   cmAnodeNgBoxLiftUpDown.monitoring.error := FALSE;
   cmAnodeNgBoxLiftUpDown.monitoring.interlockHomePos := TRUE;
   cmAnodeNgBoxLiftUpDown.monitoring.interlockWorkPos := TRUE;
   cmAnodeNgBoxLiftUpDown.monitoring.status := 16#7006;
   cmAnodeNgBoxLiftUpDown.monitoring.interlockWarningWorkPos := FALSE;
   cmAnodeNgBoxLiftUpDown.monitoring.interlockWarningHomePos := FALSE;
   cmAnodeNgBoxLiftUpDown.configuration.referenceDesignator := WSTRING#'TwoWayAct.';
   cmAnodeNgBoxLiftUpDown.configuration.monitoringLeavingFeedback := T#5S;
   cmAnodeNgBoxLiftUpDown.configuration.monitoringReachingFeedback := T#5S;
   cmAnodeNgBoxLiftUpDown.configuration.monitoringDiscrepancy := T#0MS;
   cmAnodeNgBoxLiftUpDown.configuration.setOutputHomeContinuously := TRUE;
   cmAnodeNgBoxLiftUpDown.configuration.setOutputWorkContinuously := TRUE;
   cmAnodeNgBoxLiftUpDown.configuration.disableHomeCommand := FALSE;
   cmAnodeNgBoxLiftUpDown.configuration.disableFeedbackHomePos := FALSE;
   cmAnodeNgBoxLiftUpDown.configuration.disableFeedbackWorkPos := FALSE;
   cmAnodeNgBoxLiftUpDown.configuration.disableAlarms := FALSE;
   cmAnodeNgBoxLiftUpDown.configuration.resetOutputsOnError := FALSE;
   cmAnodeNgBoxLiftUpDown.configuration.allwaysWaitOnReachingTime := FALSE;
   cmAnodeNgBoxLockUpDown.commands.refreshConfiguration := FALSE;
   cmAnodeNgBoxLockUpDown.commands.editConfiguration := FALSE;
   cmAnodeNgBoxLockUpDown.commands.saveConfiguration := FALSE;
   cmAnodeNgBoxLockUpDown.commands.reset := FALSE;
   cmAnodeNgBoxLockUpDown.commands.commandHomePos := FALSE;
   cmAnodeNgBoxLockUpDown.commands.commandWorkPos := FALSE;
   cmAnodeNgBoxLockUpDown.monitoring.enable := TRUE;
   cmAnodeNgBoxLockUpDown.monitoring.referenceDesignator := WSTRING#'NgBoxLockUpDown';
   cmAnodeNgBoxLockUpDown.monitoring.commandHomePos := FALSE;
   cmAnodeNgBoxLockUpDown.monitoring.commandWorkPos := FALSE;
   cmAnodeNgBoxLockUpDown.monitoring.goToHomePos := FALSE;
   cmAnodeNgBoxLockUpDown.monitoring.goToWorkPos := FALSE;
   cmAnodeNgBoxLockUpDown.monitoring.inHomePos := FALSE;
   cmAnodeNgBoxLockUpDown.monitoring.inWorkPos := FALSE;
   cmAnodeNgBoxLockUpDown.monitoring.reset := FALSE;
   cmAnodeNgBoxLockUpDown.monitoring.enableManualCmds := FALSE;
   cmAnodeNgBoxLockUpDown.monitoring.error := FALSE;
   cmAnodeNgBoxLockUpDown.monitoring.interlockHomePos := TRUE;
   cmAnodeNgBoxLockUpDown.monitoring.interlockWorkPos := TRUE;
   cmAnodeNgBoxLockUpDown.monitoring.status := 16#7003;
   cmAnodeNgBoxLockUpDown.monitoring.interlockWarningWorkPos := FALSE;
   cmAnodeNgBoxLockUpDown.monitoring.interlockWarningHomePos := FALSE;
   cmAnodeNgBoxLockUpDown.configuration.referenceDesignator := WSTRING#'TwoWayAct.';
   cmAnodeNgBoxLockUpDown.configuration.monitoringLeavingFeedback := T#5S;
   cmAnodeNgBoxLockUpDown.configuration.monitoringReachingFeedback := T#5S;
   cmAnodeNgBoxLockUpDown.configuration.monitoringDiscrepancy := T#0MS;
   cmAnodeNgBoxLockUpDown.configuration.setOutputHomeContinuously := TRUE;
   cmAnodeNgBoxLockUpDown.configuration.setOutputWorkContinuously := TRUE;
   cmAnodeNgBoxLockUpDown.configuration.disableHomeCommand := FALSE;
   cmAnodeNgBoxLockUpDown.configuration.disableFeedbackHomePos := FALSE;
   cmAnodeNgBoxLockUpDown.configuration.disableFeedbackWorkPos := FALSE;
   cmAnodeNgBoxLockUpDown.configuration.disableAlarms := FALSE;
   cmAnodeNgBoxLockUpDown.configuration.resetOutputsOnError := FALSE;
   cmAnodeNgBoxLockUpDown.configuration.allwaysWaitOnReachingTime := FALSE;
   cmAnodeNgPnpVaccum.commands.refreshConfiguration := FALSE;
   cmAnodeNgPnpVaccum.commands.editConfiguration := FALSE;
   cmAnodeNgPnpVaccum.commands.saveConfiguration := FALSE;
   cmAnodeNgPnpVaccum.commands.reset := FALSE;
   cmAnodeNgPnpVaccum.commands.commandHomePos := FALSE;
   cmAnodeNgPnpVaccum.commands.commandWorkPos := FALSE;
   cmAnodeNgPnpVaccum.monitoring.enable := TRUE;
   cmAnodeNgPnpVaccum.monitoring.referenceDesignator := WSTRING#'NgPnpVaccum';
   cmAnodeNgPnpVaccum.monitoring.commandHomePos := FALSE;
   cmAnodeNgPnpVaccum.monitoring.commandWorkPos := FALSE;
   cmAnodeNgPnpVaccum.monitoring.goToHomePos := FALSE;
   cmAnodeNgPnpVaccum.monitoring.goToWorkPos := FALSE;
   cmAnodeNgPnpVaccum.monitoring.inHomePos := TRUE;
   cmAnodeNgPnpVaccum.monitoring.inWorkPos := FALSE;
   cmAnodeNgPnpVaccum.monitoring.reset := FALSE;
   cmAnodeNgPnpVaccum.monitoring.enableManualCmds := FALSE;
   cmAnodeNgPnpVaccum.monitoring.error := FALSE;
   cmAnodeNgPnpVaccum.monitoring.interlockHomePos := TRUE;
   cmAnodeNgPnpVaccum.monitoring.interlockWorkPos := TRUE;
   cmAnodeNgPnpVaccum.monitoring.status := 16#7003;
   cmAnodeNgPnpVaccum.monitoring.interlockWarningWorkPos := FALSE;
   cmAnodeNgPnpVaccum.monitoring.interlockWarningHomePos := FALSE;
   cmAnodeNgPnpVaccum.configuration.referenceDesignator := WSTRING#'TwoWayAct.';
   cmAnodeNgPnpVaccum.configuration.monitoringLeavingFeedback := T#5S;
   cmAnodeNgPnpVaccum.configuration.monitoringReachingFeedback := T#5S;
   cmAnodeNgPnpVaccum.configuration.monitoringDiscrepancy := T#0MS;
   cmAnodeNgPnpVaccum.configuration.setOutputHomeContinuously := TRUE;
   cmAnodeNgPnpVaccum.configuration.setOutputWorkContinuously := TRUE;
   cmAnodeNgPnpVaccum.configuration.disableHomeCommand := FALSE;
   cmAnodeNgPnpVaccum.configuration.disableFeedbackHomePos := FALSE;
   cmAnodeNgPnpVaccum.configuration.disableFeedbackWorkPos := FALSE;
   cmAnodeNgPnpVaccum.configuration.disableAlarms := FALSE;
   cmAnodeNgPnpVaccum.configuration.resetOutputsOnError := FALSE;
   cmAnodeNgPnpVaccum.configuration.allwaysWaitOnReachingTime := FALSE;
   cmAnodeConveyorCoverFwdBwd.commands.refreshConfiguration := FALSE;
   cmAnodeConveyorCoverFwdBwd.commands.editConfiguration := FALSE;
   cmAnodeConveyorCoverFwdBwd.commands.saveConfiguration := FALSE;
   cmAnodeConveyorCoverFwdBwd.commands.reset := FALSE;
   cmAnodeConveyorCoverFwdBwd.commands.commandHomePos := FALSE;
   cmAnodeConveyorCoverFwdBwd.commands.commandWorkPos := FALSE;
   cmAnodeConveyorCoverFwdBwd.monitoring.enable := TRUE;
   cmAnodeConveyorCoverFwdBwd.monitoring.referenceDesignator := WSTRING#'ConveyorCoverFwdBwd';
   cmAnodeConveyorCoverFwdBwd.monitoring.commandHomePos := FALSE;
   cmAnodeConveyorCoverFwdBwd.monitoring.commandWorkPos := FALSE;
   cmAnodeConveyorCoverFwdBwd.monitoring.goToHomePos := FALSE;
   cmAnodeConveyorCoverFwdBwd.monitoring.goToWorkPos := FALSE;
   cmAnodeConveyorCoverFwdBwd.monitoring.inHomePos := FALSE;
   cmAnodeConveyorCoverFwdBwd.monitoring.inWorkPos := FALSE;
   cmAnodeConveyorCoverFwdBwd.monitoring.reset := FALSE;
   cmAnodeConveyorCoverFwdBwd.monitoring.enableManualCmds := FALSE;
   cmAnodeConveyorCoverFwdBwd.monitoring.error := FALSE;
   cmAnodeConveyorCoverFwdBwd.monitoring.interlockHomePos := TRUE;
   cmAnodeConveyorCoverFwdBwd.monitoring.interlockWorkPos := TRUE;
   cmAnodeConveyorCoverFwdBwd.monitoring.status := 16#7003;
   cmAnodeConveyorCoverFwdBwd.monitoring.interlockWarningWorkPos := FALSE;
   cmAnodeConveyorCoverFwdBwd.monitoring.interlockWarningHomePos := FALSE;
   cmAnodeConveyorCoverFwdBwd.configuration.referenceDesignator := WSTRING#'TwoWayAct.';
   cmAnodeConveyorCoverFwdBwd.configuration.monitoringLeavingFeedback := T#5S;
   cmAnodeConveyorCoverFwdBwd.configuration.monitoringReachingFeedback := T#5S;
   cmAnodeConveyorCoverFwdBwd.configuration.monitoringDiscrepancy := T#0MS;
   cmAnodeConveyorCoverFwdBwd.configuration.setOutputHomeContinuously := TRUE;
   cmAnodeConveyorCoverFwdBwd.configuration.setOutputWorkContinuously := TRUE;
   cmAnodeConveyorCoverFwdBwd.configuration.disableHomeCommand := FALSE;
   cmAnodeConveyorCoverFwdBwd.configuration.disableFeedbackHomePos := FALSE;
   cmAnodeConveyorCoverFwdBwd.configuration.disableFeedbackWorkPos := FALSE;
   cmAnodeConveyorCoverFwdBwd.configuration.disableAlarms := FALSE;
   cmAnodeConveyorCoverFwdBwd.configuration.resetOutputsOnError := FALSE;
   cmAnodeConveyorCoverFwdBwd.configuration.allwaysWaitOnReachingTime := FALSE;
   cmAnodeConveyorPickUpBlower.commands.refreshConfiguration := FALSE;
   cmAnodeConveyorPickUpBlower.commands.editConfiguration := FALSE;
   cmAnodeConveyorPickUpBlower.commands.saveConfiguration := FALSE;
   cmAnodeConveyorPickUpBlower.commands.reset := FALSE;
   cmAnodeConveyorPickUpBlower.commands.commandHomePos := FALSE;
   cmAnodeConveyorPickUpBlower.commands.commandWorkPos := FALSE;
   cmAnodeConveyorPickUpBlower.monitoring.enable := TRUE;
   cmAnodeConveyorPickUpBlower.monitoring.referenceDesignator := WSTRING#'ConveyorPickUpBlower';
   cmAnodeConveyorPickUpBlower.monitoring.commandHomePos := FALSE;
   cmAnodeConveyorPickUpBlower.monitoring.commandWorkPos := FALSE;
   cmAnodeConveyorPickUpBlower.monitoring.goToHomePos := FALSE;
   cmAnodeConveyorPickUpBlower.monitoring.goToWorkPos := TRUE;
   cmAnodeConveyorPickUpBlower.monitoring.inHomePos := FALSE;
   cmAnodeConveyorPickUpBlower.monitoring.inWorkPos := TRUE;
   cmAnodeConveyorPickUpBlower.monitoring.reset := FALSE;
   cmAnodeConveyorPickUpBlower.monitoring.enableManualCmds := FALSE;
   cmAnodeConveyorPickUpBlower.monitoring.error := FALSE;
   cmAnodeConveyorPickUpBlower.monitoring.interlockHomePos := TRUE;
   cmAnodeConveyorPickUpBlower.monitoring.interlockWorkPos := TRUE;
   cmAnodeConveyorPickUpBlower.monitoring.status := 16#7006;
   cmAnodeConveyorPickUpBlower.monitoring.interlockWarningWorkPos := FALSE;
   cmAnodeConveyorPickUpBlower.monitoring.interlockWarningHomePos := FALSE;
   cmAnodeConveyorPickUpBlower.configuration.referenceDesignator := WSTRING#'TwoWayAct.';
   cmAnodeConveyorPickUpBlower.configuration.monitoringLeavingFeedback := T#5S;
   cmAnodeConveyorPickUpBlower.configuration.monitoringReachingFeedback := T#5S;
   cmAnodeConveyorPickUpBlower.configuration.monitoringDiscrepancy := T#0MS;
   cmAnodeConveyorPickUpBlower.configuration.setOutputHomeContinuously := TRUE;
   cmAnodeConveyorPickUpBlower.configuration.setOutputWorkContinuously := TRUE;
   cmAnodeConveyorPickUpBlower.configuration.disableHomeCommand := FALSE;
   cmAnodeConveyorPickUpBlower.configuration.disableFeedbackHomePos := FALSE;
   cmAnodeConveyorPickUpBlower.configuration.disableFeedbackWorkPos := FALSE;
   cmAnodeConveyorPickUpBlower.configuration.disableAlarms := FALSE;
   cmAnodeConveyorPickUpBlower.configuration.resetOutputsOnError := FALSE;
   cmAnodeConveyorPickUpBlower.configuration.allwaysWaitOnReachingTime := FALSE;
   cmAlignVisionControllerInterface.commands.stepStart := FALSE;
   cmAlignVisionControllerInterface.commands.errorAck := FALSE;
   cmAlignVisionControllerInterface.commands.dataDelete := FALSE;
   cmAlignVisionControllerInterface.monitoring.profinetInput.cmdResultStatus.cmdComplete := FALSE;
   cmAlignVisionControllerInterface.monitoring.profinetInput.cmdResultStatus.cmdError := FALSE;
   cmAlignVisionControllerInterface.monitoring.profinetInput.cmdResultStatus.cmdReady := FALSE;
   cmAlignVisionControllerInterface.monitoring.profinetInput.cmdResultStatus.resultReady := FALSE;
   cmAlignVisionControllerInterface.monitoring.profinetInput.cmdResultStatus.resultOR := FALSE;
   cmAlignVisionControllerInterface.monitoring.profinetInput.cmdResultStatus.reserved0 := FALSE;
   cmAlignVisionControllerInterface.monitoring.profinetInput.cmdResultStatus.reserved1 := FALSE;
   cmAlignVisionControllerInterface.monitoring.profinetInput.cmdResultStatus.reserved2 := FALSE;
   cmAlignVisionControllerInterface.monitoring.profinetInput.trgReadyStatus.trg1Ready := FALSE;
   cmAlignVisionControllerInterface.monitoring.profinetInput.trgReadyStatus.trg2Ready := FALSE;
   cmAlignVisionControllerInterface.monitoring.profinetInput.trgReadyStatus.trg3Ready := FALSE;
   cmAlignVisionControllerInterface.monitoring.profinetInput.trgReadyStatus.trg4Ready := FALSE;
   cmAlignVisionControllerInterface.monitoring.profinetInput.trgReadyStatus.reserved0 := FALSE;
   cmAlignVisionControllerInterface.monitoring.profinetInput.trgReadyStatus.reserved1 := FALSE;
   cmAlignVisionControllerInterface.monitoring.profinetInput.trgReadyStatus.reserved2 := FALSE;
   cmAlignVisionControllerInterface.monitoring.profinetInput.trgReadyStatus.reserved3 := FALSE;
   cmAlignVisionControllerInterface.monitoring.profinetInput.trgAckStatus.trg1Ack := FALSE;
   cmAlignVisionControllerInterface.monitoring.profinetInput.trgAckStatus.trg2Ack := FALSE;
   cmAlignVisionControllerInterface.monitoring.profinetInput.trgAckStatus.trg3Ack := FALSE;
   cmAlignVisionControllerInterface.monitoring.profinetInput.trgAckStatus.trg4Ack := FALSE;
   cmAlignVisionControllerInterface.monitoring.profinetInput.trgAckStatus.reserved0 := FALSE;
   cmAlignVisionControllerInterface.monitoring.profinetInput.trgAckStatus.reserved1 := FALSE;
   cmAlignVisionControllerInterface.monitoring.profinetInput.trgAckStatus.reserved2 := FALSE;
   cmAlignVisionControllerInterface.monitoring.profinetInput.trgAckStatus.reserved3 := FALSE;
   cmAlignVisionControllerInterface.monitoring.profinetInput.miscellaneousStatus.busy := FALSE;
   cmAlignVisionControllerInterface.monitoring.profinetInput.miscellaneousStatus.err0Status := FALSE;
   cmAlignVisionControllerInterface.monitoring.profinetInput.miscellaneousStatus.err1Status := FALSE;
   cmAlignVisionControllerInterface.monitoring.profinetInput.miscellaneousStatus.remoteReady := FALSE;
   cmAlignVisionControllerInterface.monitoring.profinetInput.miscellaneousStatus.reserved0 := FALSE;
   cmAlignVisionControllerInterface.monitoring.profinetInput.miscellaneousStatus.reserved1 := FALSE;
   cmAlignVisionControllerInterface.monitoring.profinetInput.miscellaneousStatus.reserved2 := FALSE;
   cmAlignVisionControllerInterface.monitoring.profinetInput.miscellaneousStatus.reserved3 := FALSE;
   cmAlignVisionControllerInterface.monitoring.profinetInput.assignableStatus.assignable_0 := FALSE;
   cmAlignVisionControllerInterface.monitoring.profinetInput.assignableStatus.assignable_1 := FALSE;
   cmAlignVisionControllerInterface.monitoring.profinetInput.assignableStatus.assignable_2 := FALSE;
   cmAlignVisionControllerInterface.monitoring.profinetInput.assignableStatus.assignable_3 := FALSE;
   cmAlignVisionControllerInterface.monitoring.profinetInput.assignableStatus.assignable_4 := FALSE;
   cmAlignVisionControllerInterface.monitoring.profinetInput.assignableStatus.assignable_5 := FALSE;
   cmAlignVisionControllerInterface.monitoring.profinetInput.assignableStatus.assignable_6 := FALSE;
   cmAlignVisionControllerInterface.monitoring.profinetInput.assignableStatus.assignable_7 := FALSE;
   cmAlignVisionControllerInterface.monitoring.profinetInput.assignableStatus.assignable_8 := FALSE;
   cmAlignVisionControllerInterface.monitoring.profinetInput.assignableStatus.assignable_9 := FALSE;
   cmAlignVisionControllerInterface.monitoring.profinetInput.assignableStatus.assignable_10 := FALSE;
   cmAlignVisionControllerInterface.monitoring.profinetInput.assignableStatus.assignable_11 := FALSE;
   cmAlignVisionControllerInterface.monitoring.profinetInput.assignableStatus.assignable_12 := FALSE;
   cmAlignVisionControllerInterface.monitoring.profinetInput.assignableStatus.assignable_13 := FALSE;
   cmAlignVisionControllerInterface.monitoring.profinetInput.assignableStatus.assignable_14 := FALSE;
   cmAlignVisionControllerInterface.monitoring.profinetInput.assignableStatus.assignable_15 := FALSE;
   cmAlignVisionControllerInterface.monitoring.profinetInput.assignableStatus.assignable_16 := FALSE;
   cmAlignVisionControllerInterface.monitoring.profinetInput.assignableStatus.assignable_17 := FALSE;
   cmAlignVisionControllerInterface.monitoring.profinetInput.assignableStatus.assignable_18 := FALSE;
   cmAlignVisionControllerInterface.monitoring.profinetInput.assignableStatus.assignable_19 := FALSE;
   cmAlignVisionControllerInterface.monitoring.profinetInput.assignableStatus.assignable_20 := FALSE;
   cmAlignVisionControllerInterface.monitoring.profinetInput.assignableStatus.assignable_21 := FALSE;
   cmAlignVisionControllerInterface.monitoring.profinetInput.assignableStatus.assignable_22 := FALSE;
   cmAlignVisionControllerInterface.monitoring.profinetInput.assignableStatus.assignable_23 := FALSE;
   cmAlignVisionControllerInterface.monitoring.profinetInput.assignableStatus.assignable_24 := FALSE;
   cmAlignVisionControllerInterface.monitoring.profinetInput.assignableStatus.assignable_25 := FALSE;
   cmAlignVisionControllerInterface.monitoring.profinetInput.assignableStatus.assignable_26 := FALSE;
   cmAlignVisionControllerInterface.monitoring.profinetInput.assignableStatus.assignable_27 := FALSE;
   cmAlignVisionControllerInterface.monitoring.profinetInput.assignableStatus.assignable_28 := FALSE;
   cmAlignVisionControllerInterface.monitoring.profinetInput.assignableStatus.assignable_29 := FALSE;
   cmAlignVisionControllerInterface.monitoring.profinetInput.assignableStatus.assignable_30 := FALSE;
   cmAlignVisionControllerInterface.monitoring.profinetInput.assignableStatus.assignable_31 := FALSE;
   cmAlignVisionControllerInterface.monitoring.profinetInput.resultData248Byte_1.error0Code := 0;
   cmAlignVisionControllerInterface.monitoring.profinetInput.resultData248Byte_1.error1Code := 0;
   cmAlignVisionControllerInterface.monitoring.profinetInput.resultData248Byte_1.reserved12 := 0;
   cmAlignVisionControllerInterface.monitoring.profinetInput.resultData248Byte_1.totalCount := 0;
   cmAlignVisionControllerInterface.monitoring.profinetInput.resultData248Byte_1.commandResult := 0;
   cmAlignVisionControllerInterface.monitoring.profinetInput.resultData248Byte_1.commandData[0..23] := 0;
   cmAlignVisionControllerInterface.monitoring.profinetInput.resultData248Byte_1.resultData[0..33] := 0;
   cmAlignVisionControllerInterface.monitoring.profinetInput.resultData248Byte_2[0..61] := 0;
   cmAlignVisionControllerInterface.monitoring.profinetInput.resultData248Byte_3[0..61] := 0;
   cmAlignVisionControllerInterface.monitoring.profinetInput.resultData248Byte_4[0..61] := 0;
   cmAlignVisionControllerInterface.monitoring.profinetInput.resultData248Byte_5[0..61] := 0;
   cmAlignVisionControllerInterface.monitoring.profinetOutput.cmdResultControl.cmdRequest := FALSE;
   cmAlignVisionControllerInterface.monitoring.profinetOutput.cmdResultControl.inDataFbSyncInhibit := FALSE;
   cmAlignVisionControllerInterface.monitoring.profinetOutput.cmdResultControl.reserved := FALSE;
   cmAlignVisionControllerInterface.monitoring.profinetOutput.cmdResultControl.resultAck := FALSE;
   cmAlignVisionControllerInterface.monitoring.profinetOutput.cmdResultControl.err0ResetRequest := FALSE;
   cmAlignVisionControllerInterface.monitoring.profinetOutput.cmdResultControl.err1ResetRequest := FALSE;
   cmAlignVisionControllerInterface.monitoring.profinetOutput.cmdResultControl.reserved0 := FALSE;
   cmAlignVisionControllerInterface.monitoring.profinetOutput.cmdResultControl.reserved1 := FALSE;
   cmAlignVisionControllerInterface.monitoring.profinetOutput.trgControl.trg1 := FALSE;
   cmAlignVisionControllerInterface.monitoring.profinetOutput.trgControl.trg2 := FALSE;
   cmAlignVisionControllerInterface.monitoring.profinetOutput.trgControl.trg3 := FALSE;
   cmAlignVisionControllerInterface.monitoring.profinetOutput.trgControl.trg4 := FALSE;
   cmAlignVisionControllerInterface.monitoring.profinetOutput.trgControl.reserved0 := FALSE;
   cmAlignVisionControllerInterface.monitoring.profinetOutput.trgControl.reserved1 := FALSE;
   cmAlignVisionControllerInterface.monitoring.profinetOutput.trgControl.reserved2 := FALSE;
   cmAlignVisionControllerInterface.monitoring.profinetOutput.trgControl.reserved3 := FALSE;
   cmAlignVisionControllerInterface.monitoring.profinetOutput.miscellaneousControl.reset := FALSE;
   cmAlignVisionControllerInterface.monitoring.profinetOutput.miscellaneousControl.ext := FALSE;
   cmAlignVisionControllerInterface.monitoring.profinetOutput.miscellaneousControl.test := FALSE;
   cmAlignVisionControllerInterface.monitoring.profinetOutput.miscellaneousControl.reserved0 := FALSE;
   cmAlignVisionControllerInterface.monitoring.profinetOutput.miscellaneousControl.reserved1 := FALSE;
   cmAlignVisionControllerInterface.monitoring.profinetOutput.miscellaneousControl.reserved2 := FALSE;
   cmAlignVisionControllerInterface.monitoring.profinetOutput.miscellaneousControl.reserved3 := FALSE;
   cmAlignVisionControllerInterface.monitoring.profinetOutput.miscellaneousControl.reserved4 := FALSE;
   cmAlignVisionControllerInterface.monitoring.profinetOutput.reservedControl.reserved0 := FALSE;
   cmAlignVisionControllerInterface.monitoring.profinetOutput.reservedControl.reserved1 := FALSE;
   cmAlignVisionControllerInterface.monitoring.profinetOutput.reservedControl.reserved2 := FALSE;
   cmAlignVisionControllerInterface.monitoring.profinetOutput.reservedControl.reserved3 := FALSE;
   cmAlignVisionControllerInterface.monitoring.profinetOutput.reservedControl.reserved4 := FALSE;
   cmAlignVisionControllerInterface.monitoring.profinetOutput.reservedControl.reserved5 := FALSE;
   cmAlignVisionControllerInterface.monitoring.profinetOutput.reservedControl.reserved6 := FALSE;
   cmAlignVisionControllerInterface.monitoring.profinetOutput.reservedControl.reserved7 := FALSE;
   cmAlignVisionControllerInterface.monitoring.profinetOutput.assignableControl.assignable_0 := FALSE;
   cmAlignVisionControllerInterface.monitoring.profinetOutput.assignableControl.assignable_1 := FALSE;
   cmAlignVisionControllerInterface.monitoring.profinetOutput.assignableControl.assignable_2 := FALSE;
   cmAlignVisionControllerInterface.monitoring.profinetOutput.assignableControl.assignable_3 := FALSE;
   cmAlignVisionControllerInterface.monitoring.profinetOutput.assignableControl.assignable_4 := FALSE;
   cmAlignVisionControllerInterface.monitoring.profinetOutput.assignableControl.assignable_5 := FALSE;
   cmAlignVisionControllerInterface.monitoring.profinetOutput.assignableControl.assignable_6 := FALSE;
   cmAlignVisionControllerInterface.monitoring.profinetOutput.assignableControl.assignable_7 := FALSE;
   cmAlignVisionControllerInterface.monitoring.profinetOutput.assignableControl.assignable_8 := FALSE;
   cmAlignVisionControllerInterface.monitoring.profinetOutput.assignableControl.assignable_9 := FALSE;
   cmAlignVisionControllerInterface.monitoring.profinetOutput.assignableControl.assignable_10 := FALSE;
   cmAlignVisionControllerInterface.monitoring.profinetOutput.assignableControl.assignable_11 := FALSE;
   cmAlignVisionControllerInterface.monitoring.profinetOutput.assignableControl.assignable_12 := FALSE;
   cmAlignVisionControllerInterface.monitoring.profinetOutput.assignableControl.assignable_13 := FALSE;
   cmAlignVisionControllerInterface.monitoring.profinetOutput.assignableControl.assignable_14 := FALSE;
   cmAlignVisionControllerInterface.monitoring.profinetOutput.assignableControl.assignable_15 := FALSE;
   cmAlignVisionControllerInterface.monitoring.profinetOutput.assignableControl.assignable_16 := FALSE;
   cmAlignVisionControllerInterface.monitoring.profinetOutput.assignableControl.assignable_17 := FALSE;
   cmAlignVisionControllerInterface.monitoring.profinetOutput.assignableControl.assignable_18 := FALSE;
   cmAlignVisionControllerInterface.monitoring.profinetOutput.assignableControl.assignable_19 := FALSE;
   cmAlignVisionControllerInterface.monitoring.profinetOutput.assignableControl.assignable_20 := FALSE;
   cmAlignVisionControllerInterface.monitoring.profinetOutput.assignableControl.assignable_21 := FALSE;
   cmAlignVisionControllerInterface.monitoring.profinetOutput.assignableControl.assignable_22 := FALSE;
   cmAlignVisionControllerInterface.monitoring.profinetOutput.assignableControl.assignable_23 := FALSE;
   cmAlignVisionControllerInterface.monitoring.profinetOutput.assignableControl.assignable_24 := FALSE;
   cmAlignVisionControllerInterface.monitoring.profinetOutput.assignableControl.assignable_25 := FALSE;
   cmAlignVisionControllerInterface.monitoring.profinetOutput.assignableControl.assignable_26 := FALSE;
   cmAlignVisionControllerInterface.monitoring.profinetOutput.assignableControl.assignable_27 := FALSE;
   cmAlignVisionControllerInterface.monitoring.profinetOutput.assignableControl.assignable_28 := FALSE;
   cmAlignVisionControllerInterface.monitoring.profinetOutput.assignableControl.assignable_29 := FALSE;
   cmAlignVisionControllerInterface.monitoring.profinetOutput.assignableControl.assignable_30 := FALSE;
   cmAlignVisionControllerInterface.monitoring.profinetOutput.assignableControl.assignable_31 := FALSE;
   cmAlignVisionControllerInterface.monitoring.profinetOutput.parameterData248Byte_1.reversed0 := 0;
   cmAlignVisionControllerInterface.monitoring.profinetOutput.parameterData248Byte_1.reserved1 := 0;
   cmAlignVisionControllerInterface.monitoring.profinetOutput.parameterData248Byte_1.commandNumber := 0;
   cmAlignVisionControllerInterface.monitoring.profinetOutput.parameterData248Byte_1.cmdParameter[0..15] := 0;
   cmAlignVisionControllerInterface.monitoring.profinetOutput.parameterData248Byte_1.inDataFieldbus[0..42] := 0;
   cmAlignVisionControllerInterface.monitoring.profinetOutput.parameterData248Byte_2[0..61] := 0;
   cmAlignVisionControllerInterface.monitoring.profinetOutput.parameterData248Byte_3[0..61] := 0;
   cmAlignVisionControllerInterface.monitoring.profinetOutput.parameterData248Byte_4[0..61] := 0;
   cmAlignVisionControllerInterface.monitoring.profinetOutput.parameterData248Byte_5[0..61] := 0;
   cmAlignVisionControllerInterface.monitoring.resultOK := FALSE;
   cmAlignVisionControllerInterface.monitoring.resultNG := FALSE;
   cmAlignVisionControllerInterface.monitoring.resultBusy := FALSE;
   cmAlignVisionControllerInterface.monitoring.resultComplete := FALSE;
   cmAlignVisionControllerInterface.monitoring.resultData.resultData136Byte_1[0..33] := 0;
   cmAlignVisionControllerInterface.monitoring.resultData.resultData248Byte_2[0..61] := 0;
   cmAlignVisionControllerInterface.monitoring.resultData.resultData248Byte_3[0..61] := 0;
   cmAlignVisionControllerInterface.monitoring.resultData.resultData248Byte_4[0..61] := 0;
   cmAlignVisionControllerInterface.monitoring.resultData.resultData248Byte_5[0..61] := 0;
   cmAlignVisionControllerInterface.monitoring.error := FALSE;
   cmAlignVisionControllerInterface.monitoring.status := 16#0000;
   cmAlignVisionControllerInterface.configuration.hwID.cmdResultStatusID := 0;
   cmAlignVisionControllerInterface.configuration.hwID.trgReadyStatusID := 0;
   cmAlignVisionControllerInterface.configuration.hwID.trgAckStatusID := 0;
   cmAlignVisionControllerInterface.configuration.hwID.miscellaneousStatusID := 0;
   cmAlignVisionControllerInterface.configuration.hwID.assignableStatusID := 0;
   cmAlignVisionControllerInterface.configuration.hwID.resultData248ByteID_1 := 0;
   cmAlignVisionControllerInterface.configuration.hwID.resultData248ByteID_2 := 0;
   cmAlignVisionControllerInterface.configuration.hwID.resultData248ByteID_3 := 0;
   cmAlignVisionControllerInterface.configuration.hwID.resultData248ByteID_4 := 0;
   cmAlignVisionControllerInterface.configuration.hwID.resultData248ByteID_5 := 0;
   cmAlignVisionControllerInterface.configuration.hwID.cmdResultControlID := 0;
   cmAlignVisionControllerInterface.configuration.hwID.trgControlID := 0;
   cmAlignVisionControllerInterface.configuration.hwID.miscellaneousControlID := 0;
   cmAlignVisionControllerInterface.configuration.hwID.reservedControlID := 0;
   cmAlignVisionControllerInterface.configuration.hwID.assignableControlID := 0;
   cmAlignVisionControllerInterface.configuration.hwID.parameterData248ByteID_1 := 0;
   cmAlignVisionControllerInterface.configuration.hwID.parameterData248ByteID_2 := 0;
   cmAlignVisionControllerInterface.configuration.hwID.parameterData248ByteID_3 := 0;
   cmAlignVisionControllerInterface.configuration.hwID.parameterData248ByteID_4 := 0;
   cmAlignVisionControllerInterface.configuration.hwID.parameterData248ByteID_5 := 0;
   cmAlignVisionControllerInterface.configuration.referenceDesignator := WSTRING#'';
   cmAlignVisionControllerInterface.configuration.disableAlarms := FALSE;
   cmAlignVisionControllerInterface.configuration.trigger1Use := FALSE;
   cmAlignVisionControllerInterface.configuration.trigger2Use := FALSE;
   cmAlignVisionControllerInterface.configuration.trigger3Use := FALSE;
   cmAlignVisionControllerInterface.configuration.trigger4Use := FALSE;
   cmAlignVisionControllerInterface.configuration.triggertime := T#0MS;
   cmAlignVisionControllerInterface.configuration.cycleTime := T#0MS;
   cmAlignVisionControllerInterface.configuration.DataConfig.cmdResultControl.cmdRequest := FALSE;
   cmAlignVisionControllerInterface.configuration.DataConfig.cmdResultControl.inDataFbSyncInhibit := FALSE;
   cmAlignVisionControllerInterface.configuration.DataConfig.cmdResultControl.reserved := FALSE;
   cmAlignVisionControllerInterface.configuration.DataConfig.cmdResultControl.resultAck := FALSE;
   cmAlignVisionControllerInterface.configuration.DataConfig.cmdResultControl.err0ResetRequest := FALSE;
   cmAlignVisionControllerInterface.configuration.DataConfig.cmdResultControl.err1ResetRequest := FALSE;
   cmAlignVisionControllerInterface.configuration.DataConfig.cmdResultControl.reserved0 := FALSE;
   cmAlignVisionControllerInterface.configuration.DataConfig.cmdResultControl.reserved1 := FALSE;
   cmAlignVisionControllerInterface.configuration.DataConfig.trgControl.trg1 := FALSE;
   cmAlignVisionControllerInterface.configuration.DataConfig.trgControl.trg2 := FALSE;
   cmAlignVisionControllerInterface.configuration.DataConfig.trgControl.trg3 := FALSE;
   cmAlignVisionControllerInterface.configuration.DataConfig.trgControl.trg4 := FALSE;
   cmAlignVisionControllerInterface.configuration.DataConfig.trgControl.reserved0 := FALSE;
   cmAlignVisionControllerInterface.configuration.DataConfig.trgControl.reserved1 := FALSE;
   cmAlignVisionControllerInterface.configuration.DataConfig.trgControl.reserved2 := FALSE;
   cmAlignVisionControllerInterface.configuration.DataConfig.trgControl.reserved3 := FALSE;
   cmAlignVisionControllerInterface.configuration.DataConfig.miscellaneousControl.reset := FALSE;
   cmAlignVisionControllerInterface.configuration.DataConfig.miscellaneousControl.ext := FALSE;
   cmAlignVisionControllerInterface.configuration.DataConfig.miscellaneousControl.test := FALSE;
   cmAlignVisionControllerInterface.configuration.DataConfig.miscellaneousControl.reserved0 := FALSE;
   cmAlignVisionControllerInterface.configuration.DataConfig.miscellaneousControl.reserved1 := FALSE;
   cmAlignVisionControllerInterface.configuration.DataConfig.miscellaneousControl.reserved2 := FALSE;
   cmAlignVisionControllerInterface.configuration.DataConfig.miscellaneousControl.reserved3 := FALSE;
   cmAlignVisionControllerInterface.configuration.DataConfig.miscellaneousControl.reserved4 := FALSE;
   cmAlignVisionControllerInterface.configuration.DataConfig.reservedControl.reserved0 := FALSE;
   cmAlignVisionControllerInterface.configuration.DataConfig.reservedControl.reserved1 := FALSE;
   cmAlignVisionControllerInterface.configuration.DataConfig.reservedControl.reserved2 := FALSE;
   cmAlignVisionControllerInterface.configuration.DataConfig.reservedControl.reserved3 := FALSE;
   cmAlignVisionControllerInterface.configuration.DataConfig.reservedControl.reserved4 := FALSE;
   cmAlignVisionControllerInterface.configuration.DataConfig.reservedControl.reserved5 := FALSE;
   cmAlignVisionControllerInterface.configuration.DataConfig.reservedControl.reserved6 := FALSE;
   cmAlignVisionControllerInterface.configuration.DataConfig.reservedControl.reserved7 := FALSE;
   cmAlignVisionControllerInterface.configuration.DataConfig.assignableControl.assignable_0 := FALSE;
   cmAlignVisionControllerInterface.configuration.DataConfig.assignableControl.assignable_1 := FALSE;
   cmAlignVisionControllerInterface.configuration.DataConfig.assignableControl.assignable_2 := FALSE;
   cmAlignVisionControllerInterface.configuration.DataConfig.assignableControl.assignable_3 := FALSE;
   cmAlignVisionControllerInterface.configuration.DataConfig.assignableControl.assignable_4 := FALSE;
   cmAlignVisionControllerInterface.configuration.DataConfig.assignableControl.assignable_5 := FALSE;
   cmAlignVisionControllerInterface.configuration.DataConfig.assignableControl.assignable_6 := FALSE;
   cmAlignVisionControllerInterface.configuration.DataConfig.assignableControl.assignable_7 := FALSE;
   cmAlignVisionControllerInterface.configuration.DataConfig.assignableControl.assignable_8 := FALSE;
   cmAlignVisionControllerInterface.configuration.DataConfig.assignableControl.assignable_9 := FALSE;
   cmAlignVisionControllerInterface.configuration.DataConfig.assignableControl.assignable_10 := FALSE;
   cmAlignVisionControllerInterface.configuration.DataConfig.assignableControl.assignable_11 := FALSE;
   cmAlignVisionControllerInterface.configuration.DataConfig.assignableControl.assignable_12 := FALSE;
   cmAlignVisionControllerInterface.configuration.DataConfig.assignableControl.assignable_13 := FALSE;
   cmAlignVisionControllerInterface.configuration.DataConfig.assignableControl.assignable_14 := FALSE;
   cmAlignVisionControllerInterface.configuration.DataConfig.assignableControl.assignable_15 := FALSE;
   cmAlignVisionControllerInterface.configuration.DataConfig.assignableControl.assignable_16 := FALSE;
   cmAlignVisionControllerInterface.configuration.DataConfig.assignableControl.assignable_17 := FALSE;
   cmAlignVisionControllerInterface.configuration.DataConfig.assignableControl.assignable_18 := FALSE;
   cmAlignVisionControllerInterface.configuration.DataConfig.assignableControl.assignable_19 := FALSE;
   cmAlignVisionControllerInterface.configuration.DataConfig.assignableControl.assignable_20 := FALSE;
   cmAlignVisionControllerInterface.configuration.DataConfig.assignableControl.assignable_21 := FALSE;
   cmAlignVisionControllerInterface.configuration.DataConfig.assignableControl.assignable_22 := FALSE;
   cmAlignVisionControllerInterface.configuration.DataConfig.assignableControl.assignable_23 := FALSE;
   cmAlignVisionControllerInterface.configuration.DataConfig.assignableControl.assignable_24 := FALSE;
   cmAlignVisionControllerInterface.configuration.DataConfig.assignableControl.assignable_25 := FALSE;
   cmAlignVisionControllerInterface.configuration.DataConfig.assignableControl.assignable_26 := FALSE;
   cmAlignVisionControllerInterface.configuration.DataConfig.assignableControl.assignable_27 := FALSE;
   cmAlignVisionControllerInterface.configuration.DataConfig.assignableControl.assignable_28 := FALSE;
   cmAlignVisionControllerInterface.configuration.DataConfig.assignableControl.assignable_29 := FALSE;
   cmAlignVisionControllerInterface.configuration.DataConfig.assignableControl.assignable_30 := FALSE;
   cmAlignVisionControllerInterface.configuration.DataConfig.assignableControl.assignable_31 := FALSE;
   cmAlignVisionControllerInterface.configuration.DataConfig.parameterData248Byte_1.reversed0 := 0;
   cmAlignVisionControllerInterface.configuration.DataConfig.parameterData248Byte_1.reserved1 := 0;
   cmAlignVisionControllerInterface.configuration.DataConfig.parameterData248Byte_1.commandNumber := 0;
   cmAlignVisionControllerInterface.configuration.DataConfig.parameterData248Byte_1.cmdParameter[0..15] := 0;
   cmAlignVisionControllerInterface.configuration.DataConfig.parameterData248Byte_1.inDataFieldbus[0..42] := 0;
   cmAlignVisionControllerInterface.configuration.DataConfig.parameterData248Byte_2[0..61] := 0;
   cmAlignVisionControllerInterface.configuration.DataConfig.parameterData248Byte_3[0..61] := 0;
   cmAlignVisionControllerInterface.configuration.DataConfig.parameterData248Byte_4[0..61] := 0;
   cmAlignVisionControllerInterface.configuration.DataConfig.parameterData248Byte_5[0..61] := 0;
   AlignVisionConversion.tabFoldingMissingJudgementResult := 0.0;
   AlignVisionConversion.electrodeLengthJudgementResult := 0.0;
   AlignVisionConversion.electrodeHeightJudgementResult := 0.0;
   AlignVisionConversion.movementAmountAxisX1 := 0.0;
   AlignVisionConversion.movementAmountAxisY1 := 0.0;
   AlignVisionConversion.movementAmountAxisY2 := 0.0;
   AlignVisionConversion.tabFoldingMissingReply := 0.0;
   AlignVisionConversion.tabFoldingMissingUpperRangeReply := 0.0;
   AlignVisionConversion.tabFoldingMissingLowerRangeReply := 0.0;
   AlignVisionConversion.electrodeLengthReply := 0.0;
   AlignVisionConversion.electrodeLengthUpperRangeReply := 0.0;
   AlignVisionConversion.electrodeLengthLowerRangeReply := 0.0;
   AlignVisionConversion.electrodeHeightReply := 0.0;
   AlignVisionConversion.electrodeHeightUpperRangeReply := 0.0;
   AlignVisionConversion.electrodeHeightLowerRangeReply := 0.0;
   AlignVisionHistory.partID[0..50] := '';
   AlignVisionHistory.productionTimestamp[0..50] := DTL#1970-01-01-00:00:00;
   AlignVisionHistory.data[0..50].VisionOk := FALSE;
   AlignVisionHistory.data[0..50].VisionNG := FALSE;
   AlignVisionHistory.data[0..50].VisionComplete := FALSE;
   AlignVisionHistory.data[0..50]."GagueR&Rtype1OK" := FALSE;
   AlignVisionHistory.data[0..50]."GagueR&Rtype1NG" := FALSE;
   AlignVisionHistory.data[0..50]."GagueR&Rtype1Complete" := FALSE;
   AlignVisionHistory.data[0..50]."GagueR&Rtype3OK" := FALSE;
   AlignVisionHistory.data[0..50]."GagueR&Rtype3NG" := FALSE;
   AlignVisionHistory.data[0..50]."GagueR&Rtype3Complete" := FALSE;
   AlignVisionHistory.data[0..50].VisionData.tabFoldingMissingJudgementResult := 0.0;
   AlignVisionHistory.data[0..50].VisionData.electrodeLengthJudgementResult := 0.0;
   AlignVisionHistory.data[0..50].VisionData.electrodeHeightJudgementResult := 0.0;
   AlignVisionHistory.data[0..50].VisionData.movementAmountAxisX1 := 0.0;
   AlignVisionHistory.data[0..50].VisionData.movementAmountAxisY1 := 0.0;
   AlignVisionHistory.data[0..50].VisionData.movementAmountAxisY2 := 0.0;
   AlignVisionHistory.data[0..50].VisionData.tabFoldingMissingReply := 0.0;
   AlignVisionHistory.data[0..50].VisionData.tabFoldingMissingUpperRangeReply := 0.0;
   AlignVisionHistory.data[0..50].VisionData.tabFoldingMissingLowerRangeReply := 0.0;
   AlignVisionHistory.data[0..50].VisionData.electrodeLengthReply := 0.0;
   AlignVisionHistory.data[0..50].VisionData.electrodeLengthUpperRangeReply := 0.0;
   AlignVisionHistory.data[0..50].VisionData.electrodeLengthLowerRangeReply := 0.0;
   AlignVisionHistory.data[0..50].VisionData.electrodeHeightReply := 0.0;
   AlignVisionHistory.data[0..50].VisionData.electrodeHeightUpperRangeReply := 0.0;
   AlignVisionHistory.data[0..50].VisionData.electrodeHeightLowerRangeReply := 0.0;
   intCondition.Axis_05.Home.HomeInterlock := FALSE;
   intCondition.Axis_05.Home.homeinterlock_error := FALSE;
   intCondition.Axis_05.Home.intout[0..9] := FALSE;
   intCondition.Axis_05.Jog.ForwardInterlockOK := FALSE;
   intCondition.Axis_05.Jog.BackwardInterlockOk := FALSE;
   intCondition.Axis_05.Jog.ForwardInterlockError := FALSE;
   intCondition.Axis_05.Jog.BackwardInterlockError := FALSE;
   intCondition.Axis_05.Jog.intOut[0..9] := FALSE;
   intCondition.Axis_05.Position.interlockOk[0..15] := FALSE;
   intCondition.Axis_05.Position.interlockError[0..15] := FALSE;
   intCondition.Axis_05.Position.intOut[0..9] := FALSE;
   intCondition.Axis_06.Home.HomeInterlock := FALSE;
   intCondition.Axis_06.Home.homeinterlock_error := FALSE;
   intCondition.Axis_06.Home.intout[0..9] := FALSE;
   intCondition.Axis_06.Jog.ForwardInterlockOK := FALSE;
   intCondition.Axis_06.Jog.BackwardInterlockOk := FALSE;
   intCondition.Axis_06.Jog.ForwardInterlockError := FALSE;
   intCondition.Axis_06.Jog.BackwardInterlockError := FALSE;
   intCondition.Axis_06.Jog.intOut[0..9] := FALSE;
   intCondition.Axis_06.Position.interlockOk[0..15] := FALSE;
   intCondition.Axis_06.Position.interlockError[0..15] := FALSE;
   intCondition.Axis_06.Position.intOut[0..9] := FALSE;
   intCondition.Axis_11.Home.HomeInterlock := FALSE;
   intCondition.Axis_11.Home.homeinterlock_error := FALSE;
   intCondition.Axis_11.Home.intout[0..9] := FALSE;
   intCondition.Axis_11.Jog.ForwardInterlockOK := FALSE;
   intCondition.Axis_11.Jog.BackwardInterlockOk := FALSE;
   intCondition.Axis_11.Jog.ForwardInterlockError := FALSE;
   intCondition.Axis_11.Jog.BackwardInterlockError := FALSE;
   intCondition.Axis_11.Jog.intOut[0..9] := FALSE;
   intCondition.Axis_11.Position.interlockOk[0..15] := FALSE;
   intCondition.Axis_11.Position.interlockError[0..15] := FALSE;
   intCondition.Axis_11.Position.intOut[0..9] := FALSE;
   intCondition.Axis_12.Home.HomeInterlock := FALSE;
   intCondition.Axis_12.Home.homeinterlock_error := FALSE;
   intCondition.Axis_12.Home.intout[0..9] := FALSE;
   intCondition.Axis_12.Jog.ForwardInterlockOK := FALSE;
   intCondition.Axis_12.Jog.BackwardInterlockOk := FALSE;
   intCondition.Axis_12.Jog.ForwardInterlockError := FALSE;
   intCondition.Axis_12.Jog.BackwardInterlockError := FALSE;
   intCondition.Axis_12.Jog.intOut[0..9] := FALSE;
   intCondition.Axis_12.Position.interlockOk[0..15] := FALSE;
   intCondition.Axis_12.Position.interlockError[0..15] := FALSE;
   intCondition.Axis_12.Position.intOut[0..9] := FALSE;
   intCondition.Axis_14.Home.HomeInterlock := FALSE;
   intCondition.Axis_14.Home.homeinterlock_error := FALSE;
   intCondition.Axis_14.Home.intout[0..9] := FALSE;
   intCondition.Axis_14.Jog.ForwardInterlockOK := FALSE;
   intCondition.Axis_14.Jog.BackwardInterlockOk := FALSE;
   intCondition.Axis_14.Jog.ForwardInterlockError := FALSE;
   intCondition.Axis_14.Jog.BackwardInterlockError := FALSE;
   intCondition.Axis_14.Jog.intOut[0..9] := FALSE;
   intCondition.Axis_14.Position.interlockOk[0..15] := FALSE;
   intCondition.Axis_14.Position.interlockError[0..15] := FALSE;
   intCondition.Axis_14.Position.intOut[0..9] := FALSE;
   intCondition.Axis_15.Home.HomeInterlock := FALSE;
   intCondition.Axis_15.Home.homeinterlock_error := FALSE;
   intCondition.Axis_15.Home.intout[0..9] := FALSE;
   intCondition.Axis_15.Jog.ForwardInterlockOK := FALSE;
   intCondition.Axis_15.Jog.BackwardInterlockOk := FALSE;
   intCondition.Axis_15.Jog.ForwardInterlockError := FALSE;
   intCondition.Axis_15.Jog.BackwardInterlockError := FALSE;
   intCondition.Axis_15.Jog.intOut[0..9] := FALSE;
   intCondition.Axis_15.Position.interlockOk[0..15] := FALSE;
   intCondition.Axis_15.Position.interlockError[0..15] := FALSE;
   intCondition.Axis_15.Position.intOut[0..9] := FALSE;
   intCondition.Axis_16.Home.HomeInterlock := FALSE;
   intCondition.Axis_16.Home.homeinterlock_error := FALSE;
   intCondition.Axis_16.Home.intout[0..9] := FALSE;
   intCondition.Axis_16.Jog.ForwardInterlockOK := FALSE;
   intCondition.Axis_16.Jog.BackwardInterlockOk := FALSE;
   intCondition.Axis_16.Jog.ForwardInterlockError := FALSE;
   intCondition.Axis_16.Jog.BackwardInterlockError := FALSE;
   intCondition.Axis_16.Jog.intOut[0..9] := FALSE;
   intCondition.Axis_16.Position.interlockOk[0..15] := FALSE;
   intCondition.Axis_16.Position.interlockError[0..15] := FALSE;
   intCondition.Axis_16.Position.intOut[0..9] := FALSE;
   intCondition.Axis_17.Home.HomeInterlock := FALSE;
   intCondition.Axis_17.Home.homeinterlock_error := FALSE;
   intCondition.Axis_17.Home.intout[0..9] := FALSE;
   intCondition.Axis_17.Jog.ForwardInterlockOK := FALSE;
   intCondition.Axis_17.Jog.BackwardInterlockOk := FALSE;
   intCondition.Axis_17.Jog.ForwardInterlockError := FALSE;
   intCondition.Axis_17.Jog.BackwardInterlockError := FALSE;
   intCondition.Axis_17.Jog.intOut[0..9] := FALSE;
   intCondition.Axis_17.Position.interlockOk[0..15] := FALSE;
   intCondition.Axis_17.Position.interlockError[0..15] := FALSE;
   intCondition.Axis_17.Position.intOut[0..9] := FALSE;
   intCondition.Actuator_13.Home_INT := FALSE;
   intCondition.Actuator_13.Work_INT := FALSE;
   intCondition.Actuator_13.Home_INT_Error := FALSE;
   intCondition.Actuator_13.Work_INT_Error := FALSE;
   intCondition.Actuator_13.intOut[0..9] := FALSE;
   intCondition.Actuator_14.Home_INT := FALSE;
   intCondition.Actuator_14.Work_INT := FALSE;
   intCondition.Actuator_14.Home_INT_Error := FALSE;
   intCondition.Actuator_14.Work_INT_Error := FALSE;
   intCondition.Actuator_14.intOut[0..9] := FALSE;
   intCondition.Actuator_15.Home_INT := FALSE;
   intCondition.Actuator_15.Work_INT := FALSE;
   intCondition.Actuator_15.Home_INT_Error := FALSE;
   intCondition.Actuator_15.Work_INT_Error := FALSE;
   intCondition.Actuator_15.intOut[0..9] := FALSE;
   intCondition.Actuator_16.Home_INT := FALSE;
   intCondition.Actuator_16.Work_INT := FALSE;
   intCondition.Actuator_16.Home_INT_Error := FALSE;
   intCondition.Actuator_16.Work_INT_Error := FALSE;
   intCondition.Actuator_16.intOut[0..9] := FALSE;
   intCondition.Actuator_17.Home_INT := FALSE;
   intCondition.Actuator_17.Work_INT := FALSE;
   intCondition.Actuator_17.Home_INT_Error := FALSE;
   intCondition.Actuator_17.Work_INT_Error := FALSE;
   intCondition.Actuator_17.intOut[0..9] := FALSE;
   intCondition.Actuator_18.Home_INT := FALSE;
   intCondition.Actuator_18.Work_INT := FALSE;
   intCondition.Actuator_18.Home_INT_Error := FALSE;
   intCondition.Actuator_18.Work_INT_Error := FALSE;
   intCondition.Actuator_18.intOut[0..9] := FALSE;
   intCondition.Actuator_19.Home_INT := FALSE;
   intCondition.Actuator_19.Work_INT := FALSE;
   intCondition.Actuator_19.Home_INT_Error := FALSE;
   intCondition.Actuator_19.Work_INT_Error := FALSE;
   intCondition.Actuator_19.intOut[0..9] := FALSE;
   intCondition.Actuator_20.Home_INT := FALSE;
   intCondition.Actuator_20.Work_INT := FALSE;
   intCondition.Actuator_20.Home_INT_Error := FALSE;
   intCondition.Actuator_20.Work_INT_Error := FALSE;
   intCondition.Actuator_20.intOut[0..9] := FALSE;
   intCondition.Actuator_21.Home_INT := FALSE;
   intCondition.Actuator_21.Work_INT := FALSE;
   intCondition.Actuator_21.Home_INT_Error := FALSE;
   intCondition.Actuator_21.Work_INT_Error := FALSE;
   intCondition.Actuator_21.intOut[0..9] := FALSE;
   intCondition.Actuator_22.Home_INT := FALSE;
   intCondition.Actuator_22.Work_INT := FALSE;
   intCondition.Actuator_22.Home_INT_Error := FALSE;
   intCondition.Actuator_22.Work_INT_Error := FALSE;
   intCondition.Actuator_22.intOut[0..9] := FALSE;
END_DATA_BLOCK
